{attribute 'pack_mode' := '2'}
TYPE ST_GEAR_IN_MULTIMASTER :
STRUCT  
  byAxisIDMaster1  : BYTE; // AxisID of Master1
  byAxisIDMaster2  : BYTE; // AxisID of Master2
  byAxisIDMaster3  : BYTE; // AxisID of Master3
  byAxisIDMaster4  : BYTE; // AxisID of Master4
  GearRatio1       : REAL; 
  GearRatio2       : REAL; 
  GearRatio3       : REAL; 
  GearRatio4       : REAL; 
  Acceleration     : REAL;
  Deceleration     : REAL;
  Jerk             : REAL;  
END_STRUCT
END_TYPE

(* stored: Version 1.1.0.1, ProductVersion 3.1.4024.12
   DUT ST_GEAR_IN_MULTIMASTER: Id {4efdd300-d04e-0b13-188d-d85306bab98e} *)
